PROGRAM PRG_TEST
VAR
	FakeAxisContractTests : FB_FakeAxis_BaseUnitTests;
	
	MoveAbsServiceTests : FB_Chamber1SpinAxisMoveAbsServiceTests;
	MoveVelServiceTests : FB_Chamber1MoveVelServiceTests;
	
	Chamber1ModuleTests : FB_Chamber1_ModuleTests;
END_VAR

TcUnit.RUN();

END_PROGRAM

(* stored: Version 1.1.0.1, ProductVersion 3.1.4026.18
   POU PRG_TEST: Id {dd0c9370-fdb3-4448-9242-43ea44c7b9f9}, SpecialFunc None *)
